(* PLC project hopper, Dassault Systèmes ControlBuild 2024x *)
(* stored: creationDateTime 2023-10-03T11:12:59-01:00 *)

(* This module simulates the behaviour of a hopper which computes the weight and volume of material according to volumes of material that are received and substracted. *)
FUNCTION_BLOCK equipment_library.hopper
  VAR_INPUT
    volumeExtraction : REAL := 0.0;
    volumeFilling : REAL := 0.0;
    densityInput : REAL := 1.0;
  END_VAR
  VAR_OUTPUT
    levelHopper : REAL := 0.0;
    densityOutput : REAL := 0.0;
    weight : REAL := 0.0;
    percentLevel : REAL := 0.0;
    volumeOutput : REAL := 0.0;
  END_VAR
  VAR
    density : REAL := 0.0;
    realLevel : REAL := 0.0;
    debug : REAL := 0.0;
  END_VAR
  VAR CONSTANT
    capacity : REAL := 250.0;
  END_VAR
  VAR
    d_level : BOOL := false;
    v_d_level : REAL := 0.0;
  END_VAR


ACTION C_source_code:
/* -----------------------------------------------------------------	*/
/* Type : Model of Operative Behaviour					*/
/* Catégorie :   batch							*/
/* Author : Dassault Systemes						*/
/* Update date : June 2018							*/
/* -----------------------------------------------------------------	*/
/* This module simulates the behaviour of a hopper.			*/
/* The hopper computes the weight and the volume of material		*/
/* according to the volumes of received and extracted material	*/
/* ----------------------------------------------------------------	*/


/* ---------------------------------------------*/
/* compute realLevel 				*/
/* ---------------------------------------------*/
if (density == 0.0)
	density = densityInput;

realLevel += volumeFilling;   /* Physical level after filling */

if (realLevel > capacity)   realLevel = capacity;
if (realLevel < 0.0) realLevel = 0.0;
if (d_level)   levelHopper = v_d_level;
else  levelHopper += volumeFilling  - volumeExtraction;


if (levelHopper > capacity)  levelHopper = capacity;
if (levelHopper < 0.0) levelHopper = 0.0;

/* -------------------------------------------- */
/* percent of capacity 				*/
/* -------------------------------------------- */
if ( capacity!=0.0) percentLevel = levelHopper / capacity * 100.0;


if(volumeExtraction !=0.0) {
         if( (volumeExtraction <=realLevel)&&(realLevel !=0.0))  {
               volumeOutput=volumeExtraction;
         }
         else {
                volumeOutput=realLevel;
         }
}
else volumeOutput=0.0;

realLevel -= volumeExtraction; /* Physical level after extraction */
if (realLevel < 0.0) realLevel = 0.0;
/* -------------------------------------------- */
/* compute weight/density		 	  	*/
/* -------------------------------------------- */
weight = levelHopper * density;
densityOutput = density;

if (levelHopper == 0.0)
	density = 0.0;
END_ACTION
END_FUNCTION_BLOCK
